PROGRAM MAIN
VAR
	fbTest : FB_Test;
	
	i : INT;
	
	nTest : INT;
END_VAR

fbTest();

CASE i OF
	1: fbTest();
	
	2: fbTest(); nTest := fbTest.iRes;
END_CASE

END_PROGRAM

(* stored: Version 1.1.0.1, ProductVersion 3.1.4024.12
   POU MAIN: Id {e75f66b2-0f3b-4b4f-87b1-d2f1b9f38d80}, SpecialFunc None *)
